(************************************************************************************************)
(*							Beckhoff Automation Poland											*)
(*							FB_AX5000_Diag_MC2  v1.0											*)
(*									24.5.2011													*)
(*			Blok funkcyjny czytający podstawowe parametry serwa AX5xxx i jego błedy				*)
(*				Odczytane dane wpisuje do zmiennej typu ST_AX5000_Diag_MC2						*)
(*______________________________________________________________________________________________*)
FUNCTION_BLOCK FB_AX5000_Diag_MC2
VAR_OUTPUT
	bError					:	BOOL;
	ST_DIAG					:	ST_AX5000_Diag_MC2;
END_VAR
VAR_IN_OUT
	Axis					:	Axis_REF;
END_VAR
VAR
	fb_ReadAmplifierTemp		:	FB_SoEReadAmplifierTemperature;		(*MC2Drive*)
	fb_ReadDCBusCurrent		:	FB_SoEReadDcBusCurrent;				(*MC2Drive*)
	fb_ReadDCBusVoltage		: 	FB_SoEReadDcBusVoltage;				(*MC2Drive*)
	fb_ReadMotorTemp			:	FB_SoEReadMotorTemperature;			(*MC2Drive*)
	fb_ReadDiagMessage		:	FB_SoEReadDiagMessage;				(*MC2Drive*)
	fb_DiagNumber			:	FB_SoEReadDiagNumber;				(*MC2Drive*)
	fb_ReadDiagList			:	FB_SoEReadDiagNumberList;			(*MC2Drive*)
	fb_ReadC1Diagnostic		:	FB_SoERead;

	timer					:	TON;
	DiagList				:	ST_SoE_DiagNumList;
	bFirstCycle				:	BOOL	:=TRUE;
	sDiagnosticMessage		:	ST_SoE_STRING;
	ft1						:	F_TRIG;
	ft2						:	F_TRIG;
	ft3						:	F_TRIG;
	ft4						:	F_TRIG;
	ft5						:	F_TRIG;
	ft6						:	F_TRIG;
	ft7						:	F_TRIG;
	Watchdog				:	TON;
	Delay					:	TP;
END_VAR
VAR // added by the converter: edge detectors and wires of the graphical bodies
    _w1, _w2 : BOOL;
    _w3, _w4, _w5, _w6, _w7, _w8 : ANY;
END_VAR

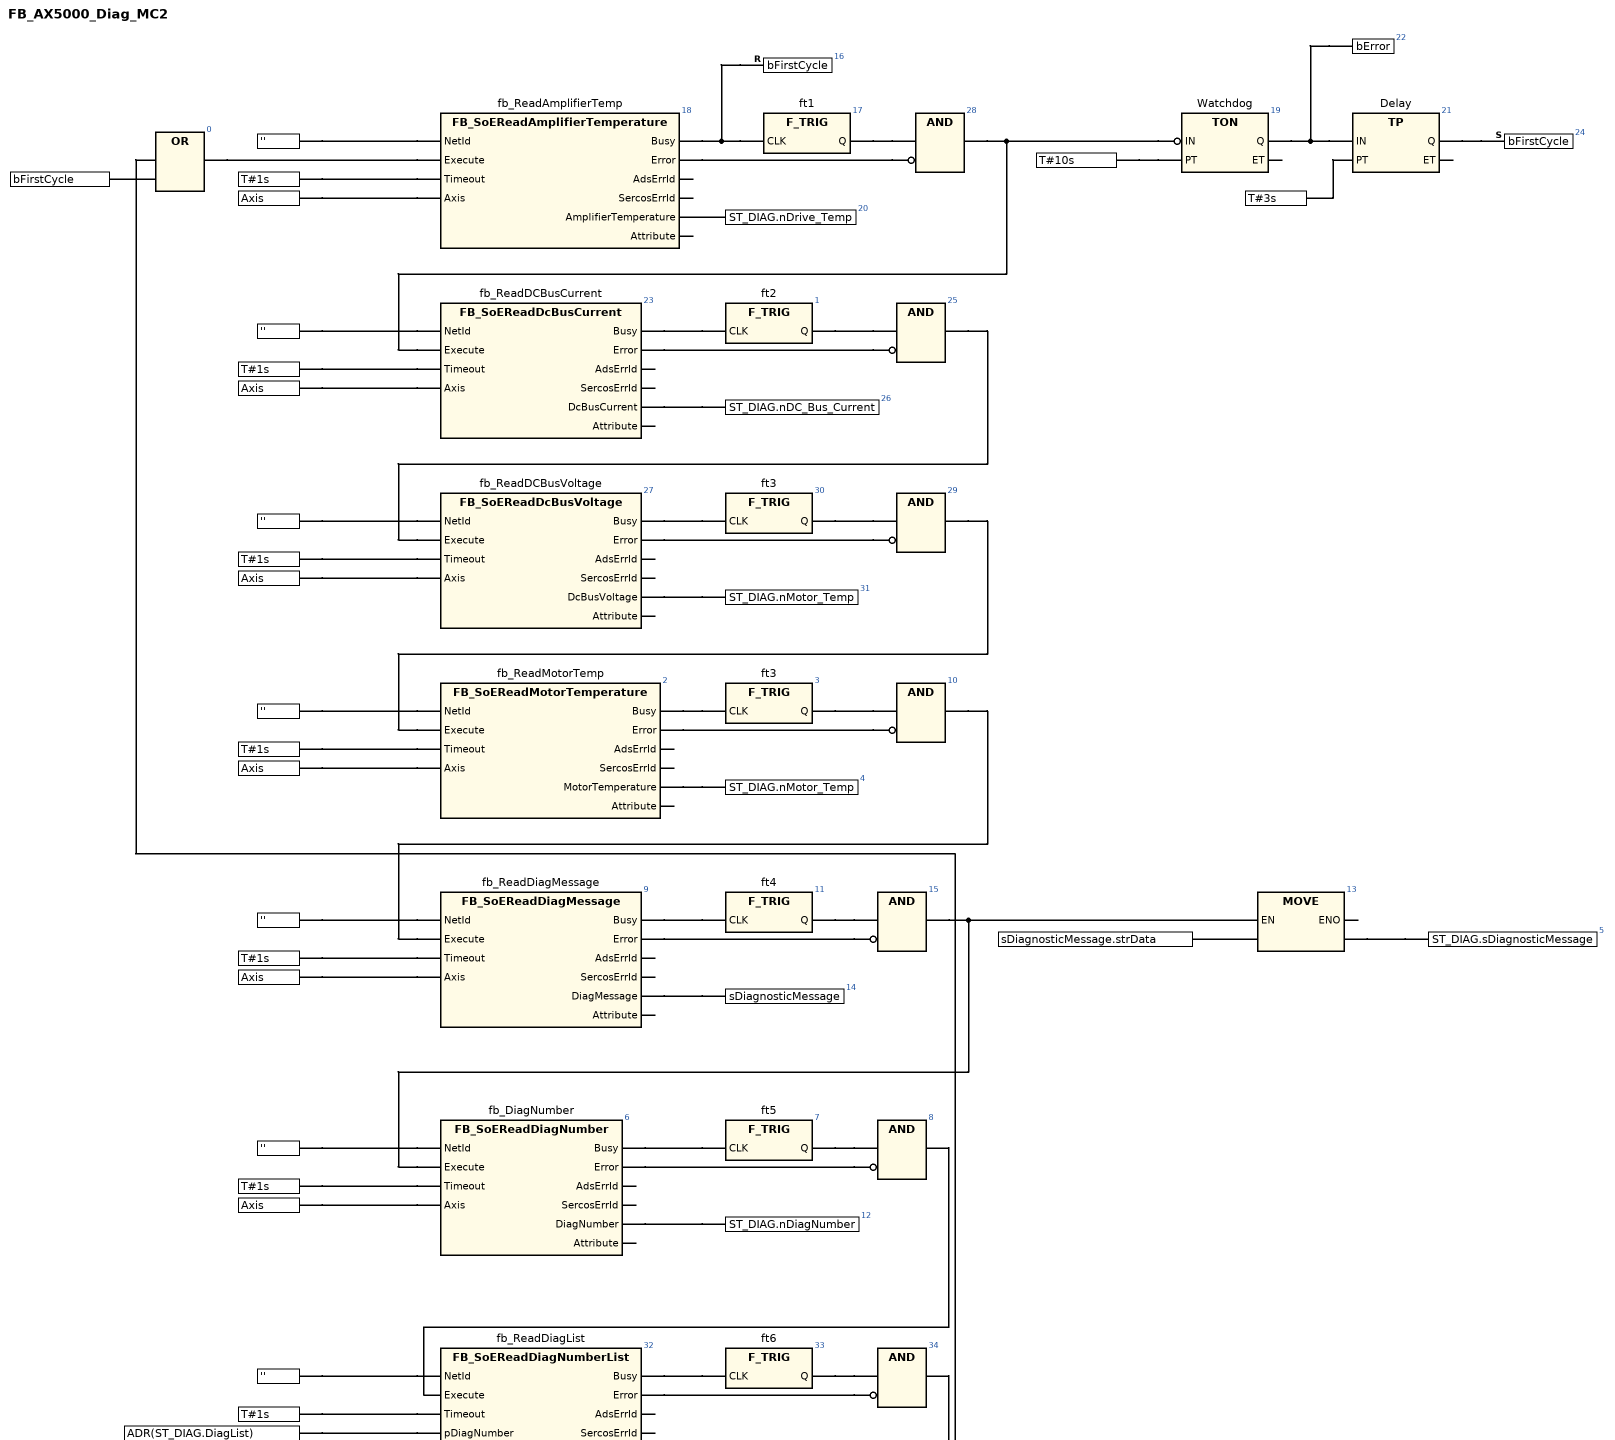
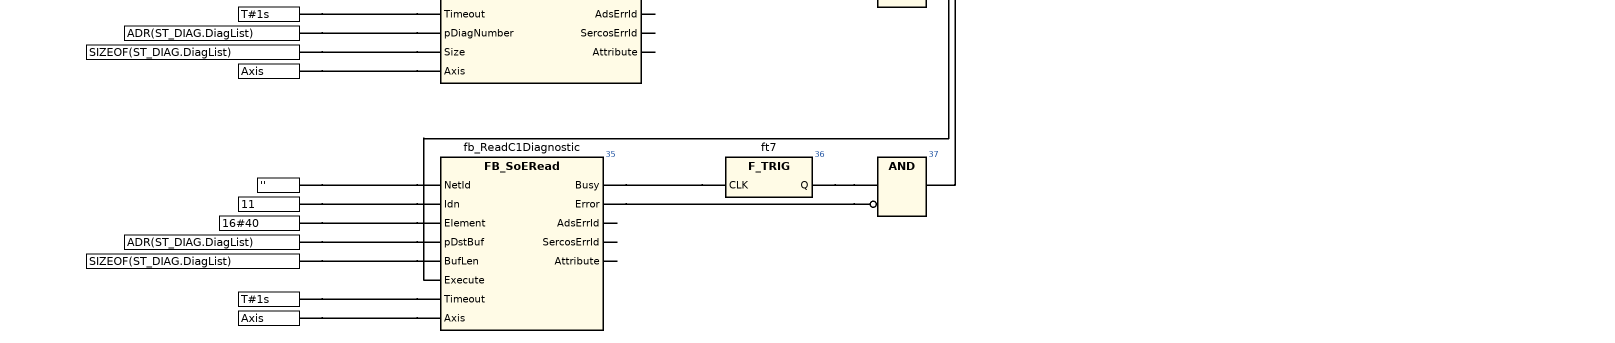
_w2 := _w1 OR bFirstCycle;
ft2(CLK := fb_ReadDCBusCurrent.Busy); // F_TRIG
fb_ReadMotorTemp(NetId := '', Execute := _w3, Timeout := T#1s, Axis := Axis); // FB_SoEReadMotorTemperature
ft3(CLK := fb_ReadMotorTemp.Busy); // F_TRIG
ST_DIAG.nMotor_Temp := fb_ReadMotorTemp.MotorTemperature;
ST_DIAG.sDiagnosticMessage := _w4;
fb_DiagNumber(NetId := '', Execute := _w5, Timeout := T#1s, Axis := Axis); // FB_SoEReadDiagNumber
ft5(CLK := fb_DiagNumber.Busy); // F_TRIG
_w6 := ft5.Q AND NOT fb_DiagNumber.Error;
fb_ReadDiagMessage(NetId := '', Execute := _w7, Timeout := T#1s, Axis := Axis); // FB_SoEReadDiagMessage
_w7 := ft3.Q AND NOT fb_ReadMotorTemp.Error;
ft4(CLK := fb_ReadDiagMessage.Busy); // F_TRIG
ST_DIAG.nDiagNumber := fb_DiagNumber.DiagNumber;
IF _w5 THEN _w4 := sDiagnosticMessage.strData; END_IF
sDiagnosticMessage := fb_ReadDiagMessage.DiagMessage;
_w5 := ft4.Q AND NOT fb_ReadDiagMessage.Error;
bFirstCycle R= fb_ReadAmplifierTemp.Busy;
ft1(CLK := fb_ReadAmplifierTemp.Busy); // F_TRIG
fb_ReadAmplifierTemp(NetId := '', Execute := _w2, Timeout := T#1s, Axis := Axis); // FB_SoEReadAmplifierTemperature
Watchdog(IN := NOT _w8, PT := T#10s); // TON
ST_DIAG.nDrive_Temp := fb_ReadAmplifierTemp.AmplifierTemperature;
Delay(IN := Watchdog.Q, PT := T#3s); // TP
bError := Watchdog.Q;
fb_ReadDCBusCurrent(NetId := '', Execute := _w8, Timeout := T#1s, Axis := Axis); // FB_SoEReadDcBusCurrent
bFirstCycle S= Delay.Q;
ST_DIAG.nDC_Bus_Current := fb_ReadDCBusCurrent.DcBusCurrent;
fb_ReadDCBusVoltage(
    NetId := '',
    Execute := ft2.Q AND NOT fb_ReadDCBusCurrent.Error,
    Timeout := T#1s,
    Axis := Axis); // FB_SoEReadDcBusVoltage
_w8 := ft1.Q AND NOT fb_ReadAmplifierTemp.Error;
_w3 := ft3.Q AND NOT fb_ReadDCBusVoltage.Error;
ft3(CLK := fb_ReadDCBusVoltage.Busy); // F_TRIG
ST_DIAG.nMotor_Temp := fb_ReadDCBusVoltage.DcBusVoltage;
fb_ReadDiagList(
    NetId := '',
    Execute := _w6,
    Timeout := T#1s,
    pDiagNumber := ADR(ST_DIAG.DiagList),
    Size := SIZEOF(ST_DIAG.DiagList),
    Axis := Axis); // FB_SoEReadDiagNumberList
ft6(CLK := fb_ReadDiagList.Busy); // F_TRIG
fb_ReadC1Diagnostic(
    NetId := '',
    Idn := 11,
    Element := 16#40,
    pDstBuf := ADR(ST_DIAG.DiagList),
    BufLen := SIZEOF(ST_DIAG.DiagList),
    Execute := ft6.Q AND NOT fb_ReadDiagList.Error,
    Timeout := T#1s,
    Axis := Axis); // FB_SoERead
ft7(CLK := fb_ReadC1Diagnostic.Busy); // F_TRIG
_w1 := ft7.Q AND NOT fb_ReadC1Diagnostic.Error;

END_FUNCTION_BLOCK

(* stored: Version 1.1.0.1, ProductVersion 3.1.4020.3
   POU FB_AX5000_Diag_MC2: Id {2e1971c9-0f6d-40cc-9d7e-38acf2eaf571}, SpecialFunc None *)
